// TIA Portal V17 export
// export: Created 2022-07-20T07:02:34.9125473Z, ExportSetting WithDefaults, DisplayName Totally Integrated Automation Portal, DisplayVersion V17, DisplayName TIA Portal Openness, DisplayVersion V17, DisplayName TIA Portal Version Control Interface, DisplayVersion V17, DisplayName SINAMICS Startdrive Advanced, DisplayVersion V17, DisplayName SINAMICS Startdrive G130, G150, S120, S150, SINAMICS MV, S210, DisplayVersion V17, DisplayName SINAMICS Startdrive G110M, G120, G120C, G120D, G120P, G115D, DisplayVersion V17, DisplayName STEP 7 Professional, DisplayVersion V17, DisplayName STEP 7 Safety, DisplayVersion V17, DisplayName WinCC Advanced, DisplayVersion V17
VAR_GLOBAL   // PLC tag table "Table de variables standard"
   P1_DI_200_0 AT %I18.0 : Bool;
   P1_DI_200_1 AT %I18.1 : Bool;
   P1_DI_200_2 AT %I18.2 : Bool;
   P1_DI_200_3 AT %I18.3 : Bool;
   P1_DI_200_4 AT %I18.4 : Bool;
   P1_DI_200_5 AT %I18.5 : Bool;
   P1_DI_200_6 AT %I18.6 : Bool;
   P1_DI_200_7 AT %I18.7 : Bool;
   P1_DI_200_8 AT %I19.0 : Bool;
   P1_DI_200_9 AT %I19.1 : Bool;
   P1_DI_200_10 AT %I19.2 : Bool;
   P1_DI_200_11 AT %I19.3 : Bool;
   P1_DI_200_12 AT %I19.4 : Bool;
   P1_DI_200_13 AT %I19.5 : Bool;
   P1_DI_200_14 AT %I19.6 : Bool;
   P1_DI_200_15 AT %I19.7 : Bool;
   P1_DI_201_0 AT %I20.0 : Bool;
   P1_DI_201_1 AT %I20.1 : Bool;
   P1_DI_201_2 AT %I20.2 : Bool;
   P1_DI_201_3 AT %I20.3 : Bool;
   P1_DI_201_4 AT %I20.4 : Bool;
   P1_DI_201_5 AT %I20.5 : Bool;
   P1_DI_201_6 AT %I20.6 : Bool;
   P1_DI_201_7 AT %I20.7 : Bool;
   P1_DI_201_8 AT %I21.0 : Bool;
   P1_DI_201_9 AT %I21.1 : Bool;
   P1_DI_201_10 AT %I21.2 : Bool;
   P1_DI_201_11 AT %I21.3 : Bool;
   P1_DI_201_12 AT %I21.4 : Bool;
   P1_DI_201_13 AT %I21.5 : Bool;
   P1_DI_201_14 AT %I21.6 : Bool;
   P1_DI_201_15 AT %I21.7 : Bool;
   P1_DQ_200_0 AT %Q8.0 : Bool;
   P1_DQ_200_1 AT %Q8.1 : Bool;
   P1_DQ_200_2 AT %Q8.2 : Bool;
   P1_DQ_200_3 AT %Q8.3 : Bool;
   P1_DQ_200_4 AT %Q8.4 : Bool;
   P1_DQ_200_5 AT %Q8.5 : Bool;
   P1_DQ_200_6 AT %Q8.6 : Bool;
   P1_DQ_200_7 AT %Q8.7 : Bool;
   P1_DQ_200_8 AT %Q9.0 : Bool;
   P1_DQ_200_9 AT %Q9.1 : Bool;
   P1_DQ_200_10 AT %Q9.2 : Bool;
   P1_DQ_200_11 AT %Q9.3 : Bool;
   P1_DQ_200_12 AT %Q9.4 : Bool;
   P1_DQ_200_13 AT %Q9.5 : Bool;
   P1_DQ_200_14 AT %Q9.6 : Bool;
   P1_DQ_200_15 AT %Q9.7 : Bool;
   P1_DQ_201_0 AT %Q10.0 : Bool;
   P1_DQ_201_1 AT %Q10.1 : Bool;
   P1_DQ_201_2 AT %Q10.2 : Bool;
   P1_DQ_201_3 AT %Q10.3 : Bool;
   P1_DQ_201_4 AT %Q10.4 : Bool;
   P1_DQ_201_5 AT %Q10.5 : Bool;
   P1_DQ_201_6 AT %Q10.6 : Bool;
   P1_DQ_201_7 AT %Q10.7 : Bool;
   P1_DQ_201_8 AT %Q11.0 : Bool;
   P1_DQ_201_9 AT %Q11.1 : Bool;
   P1_DQ_201_10 AT %Q11.2 : Bool;
   P1_DQ_201_11 AT %Q11.3 : Bool;
   P1_DQ_201_12 AT %Q11.4 : Bool;
   P1_DQ_201_13 AT %Q11.5 : Bool;
   P1_DQ_201_14 AT %Q11.6 : Bool;
   P1_DQ_201_15 AT %Q11.7 : Bool;
   P1_DQ_202_0 AT %Q12.0 : Bool;
   P1_DQ_202_1 AT %Q12.1 : Bool;
   P1_DQ_202_2 AT %Q12.2 : Bool;
   P1_DQ_202_3 AT %Q12.3 : Bool;
   P1_DQ_202_4 AT %Q12.4 : Bool;
   P1_DQ_202_5 AT %Q12.5 : Bool;
   P1_DQ_202_6 AT %Q12.6 : Bool;
   P1_DQ_202_7 AT %Q12.7 : Bool;
   P1_DQ_202_8 AT %Q13.0 : Bool;
   P1_DQ_202_9 AT %Q13.1 : Bool;
   P1_DQ_202_10 AT %Q13.2 : Bool;
   P1_DQ_202_11 AT %Q13.3 : Bool;
   P1_DQ_202_12 AT %Q13.4 : Bool;
   P1_DQ_202_13 AT %Q13.5 : Bool;
   P1_DQ_202_14 AT %Q13.6 : Bool;
   P1_DQ_202_15 AT %Q13.7 : Bool;
   P1_AI_201_0 AT %IW30 : Int;
   P1_AI_201_1 AT %IW32 : Int;
   P1_AI_201_2 AT %IW34 : Int;
   P1_AI_201_3 AT %IW36 : Int;
   P1_AI_200_1 AT %IW24 : Int;
   P1_AI_200_2 AT %IW26 : Int;
   P1_AI_200_3 AT %IW28 : Int;
   P1_AI_200_0 AT %IW22 : Int;
   P1_AI_202_0 AT %IW180 : Int;
   P1_AI_202_1 AT %IW182 : Int;
   P1_AI_202_2 AT %IW184 : Int;
   P1_AI_202_3 AT %IW186 : Int;
   P1_AQ_200_0 AT %QW168 : Int;
   P1_AQ_200_1 AT %QW170 : Int;
   P1_AQ_200_2 AT %QW172 : Int;
   P1_AQ_200_3 AT %QW174 : Int;
   P2_DI_200_0 AT %I200.0 : Bool;
   P2_DI_200_1 AT %I200.1 : Bool;
   P2_DI_200_2 AT %I200.2 : Bool;
   P2_DI_200_3 AT %I200.3 : Bool;
   P2_DI_200_4 AT %I200.4 : Bool;
   P2_DI_200_5 AT %I200.5 : Bool;
   P2_DI_200_6 AT %I200.6 : Bool;
   P2_DI_200_7 AT %I200.7 : Bool;
   P2_DI_200_8 AT %I201.0 : Bool;
   P2_DI_200_9 AT %I201.1 : Bool;
   P2_DI_200_10 AT %I201.2 : Bool;
   P2_DI_200_11 AT %I201.3 : Bool;
   P2_DI_200_12 AT %I201.4 : Bool;
   P2_DI_200_13 AT %I201.5 : Bool;
   P2_DI_200_14 AT %I201.6 : Bool;
   P2_DI_200_15 AT %I201.7 : Bool;
   P2_DI_201_0 AT %I202.0 : Bool;
   P2_DI_201_1 AT %I202.1 : Bool;
   P2_DI_201_2 AT %I202.2 : Bool;
   P2_DI_201_3 AT %I202.3 : Bool;
   P2_DI_201_4 AT %I202.4 : Bool;
   P2_DI_201_5 AT %I202.5 : Bool;
   P2_DI_201_6 AT %I202.6 : Bool;
   P2_DI_201_7 AT %I202.7 : Bool;
   P2_DI_201_8 AT %I203.0 : Bool;
   P2_DI_201_9 AT %I203.1 : Bool;
   P2_DI_201_10 AT %I203.2 : Bool;
   P2_DI_201_11 AT %I203.3 : Bool;
   P2_DI_201_12 AT %I203.4 : Bool;
   P2_DI_201_13 AT %I203.5 : Bool;
   P2_DI_201_14 AT %I203.6 : Bool;
   P2_DI_201_15 AT %I203.7 : Bool;
   P2_DQ_200_0 AT %Q200.0 : Bool;
   P2_DQ_200_1 AT %Q200.1 : Bool;
   P2_DQ_200_2 AT %Q200.2 : Bool;
   P2_DQ_200_3 AT %Q200.3 : Bool;
   P2_DQ_200_4 AT %Q200.4 : Bool;
   P2_DQ_200_5 AT %Q200.5 : Bool;
   P2_DQ_200_6 AT %Q200.6 : Bool;
   P2_DQ_200_7 AT %Q200.7 : Bool;
   P2_DQ_200_8 AT %Q201.0 : Bool;
   P2_DQ_200_9 AT %Q201.1 : Bool;
   P2_DQ_200_10 AT %Q201.2 : Bool;
   P2_DQ_200_11 AT %Q201.3 : Bool;
   P2_DQ_200_12 AT %Q201.4 : Bool;
   P2_DQ_200_13 AT %Q201.5 : Bool;
   P2_DQ_200_14 AT %Q201.6 : Bool;
   P2_DQ_200_15 AT %Q201.7 : Bool;
   P2_DQ_201_0 AT %Q202.0 : Bool;
   P2_DQ_201_1 AT %Q202.1 : Bool;
   P2_DQ_201_2 AT %Q202.2 : Bool;
   P2_DQ_201_3 AT %Q202.3 : Bool;
   P2_DQ_201_4 AT %Q202.4 : Bool;
   P2_DQ_201_5 AT %Q202.5 : Bool;
   P2_DQ_201_6 AT %Q202.6 : Bool;
   P2_DQ_201_7 AT %Q202.7 : Bool;
   P2_DQ_201_8 AT %Q203.0 : Bool;
   P2_DQ_201_9 AT %Q203.1 : Bool;
   P2_DQ_201_10 AT %Q203.2 : Bool;
   P2_DQ_201_11 AT %Q203.3 : Bool;
   P2_DQ_201_12 AT %Q203.4 : Bool;
   P2_DQ_201_13 AT %Q203.5 : Bool;
   P2_DQ_201_14 AT %Q203.6 : Bool;
   P2_DQ_201_15 AT %Q203.7 : Bool;
   P2_DQ_202_0 AT %Q204.0 : Bool;
   P2_DQ_202_1 AT %Q204.1 : Bool;
   P2_DQ_202_2 AT %Q204.2 : Bool;
   P2_DQ_202_3 AT %Q204.3 : Bool;
   P2_DQ_202_4 AT %Q204.4 : Bool;
   P2_DQ_202_5 AT %Q204.5 : Bool;
   P2_DQ_202_6 AT %Q204.6 : Bool;
   P2_DQ_202_7 AT %Q204.7 : Bool;
   P2_DQ_202_8 AT %Q205.0 : Bool;
   P2_DQ_202_9 AT %Q205.1 : Bool;
   P2_DQ_202_10 AT %Q205.2 : Bool;
   P2_DQ_202_11 AT %Q205.3 : Bool;
   P2_DQ_202_12 AT %Q205.4 : Bool;
   P2_DQ_202_13 AT %Q205.5 : Bool;
   P2_DQ_202_14 AT %Q205.6 : Bool;
   P2_DQ_202_15 AT %Q205.7 : Bool;
   P2_AI_200_0 AT %IW44 : Int;
   P2_AI_200_1 AT %IW46 : Int;
   P2_AI_200_2 AT %IW48 : Int;
   P2_AI_200_3 AT %IW50 : Int;
   P2_AI_201_0 AT %IW212 : Int;
   P2_AI_201_1 AT %IW214 : Int;
   P2_AI_201_2 AT %IW216 : Int;
   P2_AI_201_3 AT %IW218 : Int;
   P2_AI_202_0 AT %IW220 : Int;
   P2_AI_202_1 AT %IW222 : Int;
   P2_AI_202_2 AT %IW224 : Int;
   P2_AI_202_3 AT %IW226 : Int;
   P2_AQ_200_0 AT %QW206 : Int;
   P2_AQ_200_1 AT %QW208 : Int;
   P2_AQ_200_2 AT %QW210 : Int;
   P2_AQ_200_3 AT %QW212 : Int;
   TO_20000_UnwinderAxis_Actor_Interface_AddressIn AT %I516.0 : "PD_TEL105_IN";
   TO_20000_UnwinderAxis_Actor_Interface_AddressOut AT %Q516.0 : "PD_TEL105_OUT";
   TO_20000_UnwinderAxis_Actor_Interface_TorqueDataAddressIn AT %I736.0 : "PD_TEL750_IN";
   TO_20000_UnwinderAxis_Actor_Interface_TorqueDataAddressOut AT %Q736.0 : "PD_TEL750_OUT";
   TO_20001_InfeedMasterAxis_Actor_Interface_AddressIn AT %I536.0 : "PD_TEL105_IN";
   TO_20001_InfeedMasterAxis_Actor_Interface_AddressOut AT %Q536.0 : "PD_TEL105_OUT";
   TO_20001_InfeedMasterAxis_Actor_Interface_TorqueDataAddressIn AT %I742.0 : "PD_TEL750_IN";
   TO_20001_InfeedMasterAxis_Actor_Interface_TorqueDataAddressOut AT %Q742.0 : "PD_TEL750_OUT";
   TO_20002_OutfeedAxis_Actor_Interface_AddressIn AT %I556.0 : "PD_TEL105_IN";
   TO_20002_OutfeedAxis_Actor_Interface_AddressOut AT %Q556.0 : "PD_TEL105_OUT";
   TO_20002_OutfeedAxis_Actor_Interface_TorqueDataAddressIn AT %I748.0 : "PD_TEL750_IN";
   TO_20002_OutfeedAxis_Actor_Interface_TorqueDataAddressOut AT %Q748.0 : "PD_TEL750_OUT";
   TO_20003_BufferAxis_Actor_Interface_AddressIn AT %I576.0 : "PD_TEL105_IN";
   TO_20003_BufferAxis_Actor_Interface_AddressOut AT %Q576.0 : "PD_TEL105_OUT";
   TO_20003_BufferAxis_Actor_Interface_TorqueDataAddressIn AT %I754.0 : "PD_TEL750_IN";
   TO_20003_BufferAxis_Actor_Interface_TorqueDataAddressOut AT %Q754.0 : "PD_TEL750_OUT";
   TO20004_IfoilTrolley_Actor_Interface_AddressIn AT %I596.0 : "PD_TEL105_IN";
   TO20004_IfoilTrolley_Actor_Interface_AddressOut AT %Q596.0 : "PD_TEL105_OUT";
   TO20004_IfoilTrolley_Actor_Interface_TorqueDataAddressIn AT %I760.0 : "PD_TEL750_IN";
   TO20004_IfoilTrolley_Actor_Interface_TorqueDataAddressOut AT %Q760.0 : "PD_TEL750_OUT";
   TO20005_IfoilHeatingAxis_Actor_Interface_AddressIn AT %I616.0 : "PD_TEL105_IN";
   TO20005_IfoilHeatingAxis_Actor_Interface_AddressOut AT %Q616.0 : "PD_TEL105_OUT";
   TO20005_IfoilHeatingAxis_Actor_Interface_TorqueDataAddressIn AT %I766.0 : "PD_TEL750_IN";
   TO20005_IfoilHeatingAxis_Actor_Interface_TorqueDataAddressOut AT %Q766.0 : "PD_TEL750_OUT";
   TO20006_IfoilInfeedAxis_Actor_Interface_AddressIn AT %I636.0 : "PD_TEL105_IN";
   TO20006_IfoilInfeedAxis_Actor_Interface_AddressOut AT %Q636.0 : "PD_TEL105_OUT";
   TO20006_IfoilInfeedAxis_Actor_Interface_TorqueDataAddressIn AT %I772.0 : "PD_TEL750_IN";
   TO20006_IfoilInfeedAxis_Actor_Interface_TorqueDataAddressOut AT %Q772.0 : "PD_TEL750_OUT";
   TO20007_IfoilOutfeedAxis_Actor_Interface_AddressIn AT %I656.0 : "PD_TEL105_IN";
   TO20007_IfoilOutfeedAxis_Actor_Interface_AddressOut AT %Q656.0 : "PD_TEL105_OUT";
   TO20007_IfoilOutfeedAxis_Actor_Interface_TorqueDataAddressIn AT %I778.0 : "PD_TEL750_IN";
   TO20007_IfoilOutfeedAxis_Actor_Interface_TorqueDataAddressOut AT %Q778.0 : "PD_TEL750_OUT";
   TO20008_InfeedRewinderAxis_Actor_Interface_AddressIn AT %I676.0 : "PD_TEL105_IN";
   TO20008_InfeedRewinderAxis_Actor_Interface_AddressOut AT %Q676.0 : "PD_TEL105_OUT";
   TO20008_InfeedRewinderAxis_Actor_Interface_TorqueDataAddressIn AT %I784.0 : "PD_TEL750_IN";
   TO20008_InfeedRewinderAxis_Actor_Interface_TorqueDataAddressOut AT %Q784.0 : "PD_TEL750_OUT";
   TO20009_Actor_Interface_AddressIn AT %I696.0 : "PD_TEL105_IN";
   TO20009_Actor_Interface_AddressOut AT %Q696.0 : "PD_TEL105_OUT";
   TO20009_Actor_Interface_TorqueDataAddressIn AT %I796.0 : "PD_TEL750_IN";
   TO20009_Actor_Interface_TorqueDataAddressOut AT %Q796.0 : "PD_TEL750_OUT";
   TO20010_RewinderTopAxis_Actor_Interface_AddressIn AT %I716.0 : "PD_TEL105_IN";
   TO20010_RewinderTopAxis_Actor_Interface_AddressOut AT %Q716.0 : "PD_TEL105_OUT";
   TO20010_RewinderTopAxis_Actor_Interface_TorqueDataAddressIn AT %I790.0 : "PD_TEL750_IN";
   TO20010_RewinderTopAxis_Actor_Interface_TorqueDataAddressOut AT %Q790.0 : "PD_TEL750_OUT";
   RewinderBottomActualTension AT %MW408 : Word;
   SMC_2_Output_1 AT %QB802 : Byte;
   SMC_2_Output_2 AT %QB803 : Byte;
   SMC_2_Output_3 AT %QB804 : Byte;
   SMC_2_Output_4 AT %QB805 : Byte;
   PTO_Axis_Actor_Interface_AddressIn AT %I841.0 : "PD_TEL1_IN";
   PTO_Axis_Actor_Interface_AddressOut AT %Q818.0 : "PD_TEL1_OUT";
   PTO_Axis_Sensor1_Interface_AddressIn AT %I845.0 : "PD_TEL81_IN";
   PTO_Axis_Sensor1_Interface_AddressOut AT %Q822.0 : "PD_TEL81_OUT";
   System_Byte AT %MB1 : Byte;
END_VAR
VAR_GLOBAL CONSTANT   // user constants
   INFEED_MASTER_AXIS : Int := 2;
   OUTFEED_AXIS : Int := 3;
   BUFFER_AXIS : Int := 4;
   IFOIL_TROLLEY_AXIS : Int := 5;
   IFOIL_HEATING_AXIS : Int := 6;
   IFOIL_INFEED_AXIS : Int := 7;
   IFOIL_OUTFEED_AXIS : Int := 8;
   INFEED_REWINDER_AXIS : Int := 9;
   REWINDER_BOTTOM_AXIS : Int := 10;
   REWINDER_TOP_AXIS : Int := 11;
   MASTER_OUTFEED_VIRTUAL_AXIS : Int := 12;
   NUMBER_OF_AXIS : Int := 13;
   UNWINDER_TECH : Int := 1;
   REWINDER_BOTTOM_TECH : Int := 2;
   REWINDER_TOP_TECH : Int := 3;
   OUTFEED_TECH : Int := 1;
   INFEED_REWINDER_TECH : Int := 2;
   "0_VIRTUAL_STATE_IDLE" : Int := 0;
   "10_VIRTUAL_STATE_ENABLE_FB" : Int := 10;
   "20_VIRTUAL_STATE_WAIT_FB_ENABLED" : Int := 20;
   "30_VIRTUAL_STATE_FB_ENABLED" : Int := 30;
   "40_VIRTUAL_STATE_ENABLE_AXIS" : Int := 40;
   "50_VIRTUAL_STATE_WAIT_AXIS_ENABLED" : Int := 50;
   "90_VIRTUAL_STATE_IN_OPERATION" : Int := 90;
   "100_VIRTUAL_STATE_START_LINE" : Int := 100;
   "110_VIRTUAL_STATE_LINE_IN_MOTION" : Int := 110;
   "120_VIRTUAL_STATE_STOP_LINE" : Int := 120;
   "130_VIRTUAL_STATE_LINE_STOPPING" : Int := 130;
   "140_VIRTUAL_STATE_LINE_STOPPED" : Int := 140;
   "200_VIRTUAL_STATE_DISABLE_AXIS" : Int := 200;
   "210_VIRTUAL_STATE_WAIT_AXIS_DISABLED" : Int := 210;
   "220_VIRTUAL_STATE_DISABLE_FB" : Int := 220;
   "230_VIRTUAL_STATE_WAIT_FB_DISABLED" : Int := 230;
   "240_VIRTUAL_STATE_FB_DISABLED" : Int := 240;
   "900_VIRTUAL_STATE_ERROR" : Int := 900;
   "60_VIRTUAL_STATE_GEARIN_RELATIVE" : Int := 60;
   "70_VIRTUAL_STATE_WAIT_IN_SYNC" : Int := 70;
   "80_VIRTUAL_STATE_IN_SYNC" : Int := 80;
   "0_BUFFER_STATE_IDLE" : Int := 0;
   "10_BUFFER_STATE_ENABLE_FB" : Int := 10;
   "20_BUFFER_STATE_WAIT_FB_ENABLED" : Int := 20;
   "30_BUFFER_STATE_FB_ENABLED" : Int := 30;
   "60_BUFFER_STATE_ENABLE_AXIS" : Int := 60;
   "70_BUFFER_STATE_WAIT_AXIS_ENABLED" : Int := 70;
   "110_BUFFER_STATE_IN_OPERATION" : Int := 110;
   "120_BUFFER_STATE_START_MOVING_TO_STOP_POS" : Int := 120;
   "130_BUFFER_STATE_IN_MOTION_TO_STOP_POS" : Int := 130;
   "150_BUFFER_STATE_STOP_BUFFER" : Int := 150;
   "160_BUFFER_STATE_BUFFER_STOPPING" : Int := 160;
   "170_BUFFER_STATE_BUFFER_STOPPED" : Int := 170;
   "180_BUFFER_STATE_DISABLE_AXIS" : Int := 180;
   "190_BUFFER_STATE_WAIT_AXIS_DISABLED" : Int := 190;
   "220_BUFFER_STATE_DISABLE_FB" : Int := 220;
   "230_BUFFER_STATE_WAIT_FB_DISABLED" : Int := 230;
   "240_BUFFER_STATE_FB_DISABLED" : Int := 240;
   "900_BUFFER_STATE_ERROR" : Int := 900;
   "80_BUFFER_STATE_MOVE_TO_START_POS" : Int := 80;
   "90_BUFFER_STATE_IN_MOTION_TO_START_POS" : Int := 90;
   "100_BUFFER_STATE_IN_START_POSITION" : Int := 100;
   "140_BUFFER_STATE_IN_STOP_POSITION" : Int := 140;
   "40_BUFFER_STATE_ACTIVE_TORQUE_LIMIT" : Int := 40;
   "50_BUFFER_STATE_TORQUE_LIMITATION_ACTIVE" : Int := 50;
   "200_BUFFER_STATE_DESACTIVE_TORQUE_LIMIT" : Int := 200;
   "210_BUFFER_STATE_TORQUE_LIMITATION_INACTIVE" : Int := 210;
   "210_LINE_STATE_IN_POSITION_REV" : Int := 210;
   PTO_AXIS : Int := 13;
   "90_LINE_STATE_WAIT_SLAVE_AXIS_IN_SYNC" : Int := 90;
   "81_BUFFER_STATE_JOG_TO_START_POS" : Int := 81;
   "91_BUFFER_STATE_IN_JOG_TO_START_POS" : Int := 91;
   "60_WINDER_STATE_FB_ENABLED" : Int := 60;
   "200_LINE_STATE_POSITIONING_REV" : Int := 200;
   "0_IFOIL_TROLLEY_STATE_IDLE" : Int := 0;
   "10_IFOIL_TROLLEY_STATE_ENABLE_FB" : Int := 10;
   "20_IFOIL_TROLLEY_STATE_WAIT_FB_ENABLED" : Int := 20;
   "30_IFOIL_TROLLEY_STATE_FB_ENABLED" : Int := 30;
   "60_IFOIL_TROLLEY_STATE_ENABLE_AXIS" : Int := 60;
   "70_IFOIL_TROLLEY_STATE_WAIT_AXIS_ENABLED" : Int := 70;
   "110_IFOIL_TROLLEY_STATE_IN_OPERATION" : Int := 110;
   "120_IFOIL_TROLLEY_STATE_START_MOVING_TO_STOP_POS" : Int := 120;
   "130_IFOIL_TROLLEY_STATE_IN_MOTION_TO_STOP_POS" : Int := 130;
   "150_IFOIL_TROLLEY_STATE_STOP_TROLLEY" : Int := 150;
   "160_IFOIL_TROLLEY_STATE_TROLLEY_STOPPING" : Int := 160;
   "170_IFOIL_TROLLEY_STATE_TROLLEY_STOPPED" : Int := 170;
   "180_IFOIL_TROLLEY_STATE_DISABLE_AXIS" : Int := 180;
   "190_IFOIL_TROLLEY_STATE_WAIT_AXIS_DISABLED" : Int := 190;
   "220_IFOIL_TROLLEY_STATE_DISABLE_FB" : Int := 220;
   "230_IFOIL_TROLLEY_STATE_WAIT_FB_DISABLED" : Int := 230;
   "240_IFOIL_TROLLEY_STATE_FB_DISABLED" : Int := 240;
   "900_IFOIL_TROLLEY_STATE_ERROR" : Int := 900;
   "80_IFOIL_TROLLEY_STATE_MOVE_TO_START_POS" : Int := 80;
   "90_IFOIL_TROLLEY_STATE_IN_MOTION_TO_START_POS" : Int := 90;
   "100_IFOIL_TROLLEY_STATE_IN_START_POSITION" : Int := 100;
   "140_IFOIL_TROLLEY_STATE_IN_STOP_POSITION" : Int := 140;
   "40_IFOIL_TROLLEY_STATE_ACTIVE_TORQUE_LIMIT" : Int := 40;
   "50_IFOIL_TROLLEY_STATE_TORQUE_LIMITATION_ACTIVE" : Int := 50;
   "200_IFOIL_TROLLEY_STATE_DESACTIVE_TORQUE_LIMIT" : Int := 200;
   "210_IFOIL_TROLLEY_STATE_TORQUE_LIMITATION_INACTIVE" : Int := 210;
   "81_IFOIL_TROLLEY_STATE_JOG_TO_START_POS" : Int := 81;
   "91_IFOIL_TROLLEY_STATE_IN_JOG_TO_START_POS" : Int := 91;
   MAX_NUMBER_OF_FOIL_AREA : UInt := 6;
   MAX_IFOIL_FIFO_ITEMS_NUMBER : UInt := 10;
   "91_VIRTUAL_STATE_CHANGE_RATIO" : Int := 91;
END_VAR
